{attribute 'reflection'}
FUNCTION_BLOCK PUBLIC FB_DevPushbuttonLight EXTENDS Fb_DevDigitalInputFunctions
VAR_OUTPUT
END_VAR
VAR
	fbLight : Fb_DevLight ; // light control 
END_VAR

// Set device type
IF eDevType = E_Devices.Undefined THEN 
	eDevType := E_Devices.PushButtonLight ;
END_IF

SUPER^(refFbFault := refFbFault);

// Light commands
	
fbLight(bEnable := bEnable, refFbFault := refFbFault);

METHOD PUBLIC CmdBlinkFast : BOOL
VAR_INPUT
END_VAR
CmdBlinkFast := fbLight.CmdBlinkFast();
END_METHOD

METHOD PUBLIC CmdBlinkSlow : BOOL
VAR_INPUT
END_VAR
CmdBlinkSlow	:= fbLight.CmdBlinkSlow();
END_METHOD

METHOD PUBLIC CmdOn : BOOL
VAR_INPUT
END_VAR
CmdOn := fbLight.CmdOn() ;
END_METHOD

END_FUNCTION_BLOCK

(* stored: Version 1.1.0.1, ProductVersion 3.1.4024.5
   POU FB_DevPushbuttonLight: Id {07fab308-52dd-4cfa-88cc-f84e729aee41}, SpecialFunc None
   Method CmdBlinkFast: Id {833ab54e-998c-06b2-361a-88ca4c5012fa}
   Method CmdBlinkSlow: Id {a3998136-c2d9-0929-2ed9-df7052e83a4f}
   Method CmdOn: Id {70490632-31ec-0540-1e03-ae338bee4da0} *)
